// TIA Portal V20 export
ORGANIZATION_BLOCK "Startup"   // OB1020, LAD, Startup
TITLE = "Complete Restart"
// stored: AutoNumber false, IsIECCheckEnabled true, Namespace Unit1.Em3, SetENOAutomatically true
   VAR_INPUT
      LostRetentive : Bool;   // True if retentive data are lost
      LostRTC : Bool;   // True if date and time are lost
   END_VAR
BEGIN

REGION Network 1 (SCL): Build the Absolut Reference Designator
   // Set the Absoult Reference Designator in the Config DB
   IF LEN(IN := "Unit1.Em3.Config".em.referenceDesignator.parent) <> 0 THEN
       "Unit1.Em3.Config".em.referenceDesignator.combined := CONCAT_WSTRING(IN1 := "Unit1.Em3.Config".em.referenceDesignator.parent, IN2 := WSTRING#'.', IN3 := "Unit1.Em3.Config".em.referenceDesignator.relative);
   ELSE
       "Unit1.Em3.Config".em.referenceDesignator.combined := "Unit1.Em3.Config".em.referenceDesignator.relative;
   END_IF;
END_REGION

REGION Network 2 (SCL): Assign axes data
   // This is an example how to assign axes to DB_ANY in DB Config. If you have axes, assign them here. The Config.axis[] variables will be handed over to the control modules. That enables a flexible programming.
   // Assign axes
   "Unit1.MotionNodes".PLCToMotion.TechnologyObject.Axis.MasterVirtual := "Unit1.Em3.Config".axis[1] := "BA010AZCR_MasterVirtualAxis";
   "Unit1.MotionNodes".PLCToMotion.TechnologyObject.Axis.UnwinderVirtual := "Unit1.Em3.Config".axis[2] := "BA010AZCR_UnwinderVirtualAxis";

   // FB Enable
   "Unit1.Em3.HmiInterface".cmMasterVirtualAxis.commands.enable := TRUE;
END_REGION

REGION Network 3 (SCL): CM Config
   // Master Virtual Axis
   "Unit1.Em3.Config".cmMasterVirtualAxis.referenceDesignator := WSTRING#'MasterVirtualAxis';
   "Unit1.Em3.Config".cmMasterVirtualAxis.disableAlarms := FALSE;
   "Unit1.Em3.Config".cmMasterVirtualAxis.masterControlPopUp := TRUE;

   // Unwinder Virtual Axis
   "Unit1.Em3.Config".cmUnwinderVirtualAxis.referenceDesignator := WSTRING#'UnwinderVirtualAxis';
   "Unit1.Em3.Config".cmUnwinderVirtualAxis.disableAlarms := FALSE;
   "Unit1.Em3.Config".cmUnwinderVirtualAxis.masterControlPopUp := TRUE;


   // Dancer Regulator
   "Unit1.Em3.Config".cmDancerRegulatorOnOff.referenceDesignator := WSTRING#'Dancer Regulator';
   "Unit1.Em3.Config".cmDancerRegulatorOnOff.monitoringLeavingFeedback := T#0MS;
   "Unit1.Em3.Config".cmDancerRegulatorOnOff.monitoringReachingFeedback := T#0MS;
   "Unit1.Em3.Config".cmDancerRegulatorOnOff.monitoringDiscrepancy := T#0ms;
   "Unit1.Em3.Config".cmDancerRegulatorOnOff.setOutputHomeContinuously := TRUE;
   "Unit1.Em3.Config".cmDancerRegulatorOnOff.setOutputWorkContinuously := TRUE;
   "Unit1.Em3.Config".cmDancerRegulatorOnOff.disableHomeCommand := FALSE;
   "Unit1.Em3.Config".cmDancerRegulatorOnOff.disableFeedbackHomePos := TRUE;
   "Unit1.Em3.Config".cmDancerRegulatorOnOff.disableFeedbackWorkPos := TRUE;
   "Unit1.Em3.Config".cmDancerRegulatorOnOff.disableAlarms := FALSE;
   "Unit1.Em3.Config".cmDancerRegulatorOnOff.resetOutputsOnError := FALSE;
   "Unit1.Em3.Config".cmDancerRegulatorOnOff.allwaysWaitOnReachingTime := FALSE;


   // Dancer Encoder
   "Unit1.Em3.Config".cmDancerEncoderAnalogInput.referenceDesignator := WSTRING#'Dancer Encoder';
   "Unit1.Em3.Config".cmDancerEncoderAnalogInput.physicalUnit := 'deg';
   "Unit1.Em3.Config".cmDancerEncoderAnalogInput.isUnipolarSignal := TRUE;
   "Unit1.Em3.Config".cmDancerEncoderAnalogInput.default := 0;
   "Unit1.Em3.Config".cmDancerEncoderAnalogInput.limitHigh2 := 20;
   "Unit1.Em3.Config".cmDancerEncoderAnalogInput.limitHigh1 := 15;
   "Unit1.Em3.Config".cmDancerEncoderAnalogInput.limitLow1 := -15;
   "Unit1.Em3.Config".cmDancerEncoderAnalogInput.limitLow2 := -20;
   "Unit1.Em3.Config".cmDancerEncoderAnalogInput.processValueMax := 43;
   "Unit1.Em3.Config".cmDancerEncoderAnalogInput.processValueMin := -43;
   "Unit1.Em3.Config".cmDancerEncoderAnalogInput.scaleAnalogUppPoint := 27648;
   "Unit1.Em3.Config".cmDancerEncoderAnalogInput.scaleAnalogLowPoint := 0;
   "Unit1.Em3.Config".cmDancerEncoderAnalogInput.scaleProcessUppPoint := 43;
   "Unit1.Em3.Config".cmDancerEncoderAnalogInput.scaleProcessLowPoint := -43;
   "Unit1.Em3.Config".cmDancerEncoderAnalogInput.disableAlarms := FALSE;


   // Dancer Electro Pneumatic Regulator
   "Unit1.Em3.Config".cmDancerElectroPneumaticRegulatorAnalogOutput.referenceDesignator := WSTRING#'Dancer Regulator';
   "Unit1.Em3.Config".cmDancerElectroPneumaticRegulatorAnalogOutput.physicalUnit := 'MPa';
   "Unit1.Em3.Config".cmDancerElectroPneumaticRegulatorAnalogOutput.isUnipolarSignal := TRUE;
   "Unit1.Em3.Config".cmDancerElectroPneumaticRegulatorAnalogOutput.default := 0;
   "Unit1.Em3.Config".cmDancerElectroPneumaticRegulatorAnalogOutput.limitHigh2 := 90;
   "Unit1.Em3.Config".cmDancerElectroPneumaticRegulatorAnalogOutput.limitHigh1 := 80;
   "Unit1.Em3.Config".cmDancerElectroPneumaticRegulatorAnalogOutput.limitLow1 := -80;
   "Unit1.Em3.Config".cmDancerElectroPneumaticRegulatorAnalogOutput.limitLow2 := -90;
   "Unit1.Em3.Config".cmDancerElectroPneumaticRegulatorAnalogOutput.processValueMax := 0.5;
   "Unit1.Em3.Config".cmDancerElectroPneumaticRegulatorAnalogOutput.processValueMin := 0.005;
   "Unit1.Em3.Config".cmDancerElectroPneumaticRegulatorAnalogOutput.scaleProcessUppPoint := 0.5;
   "Unit1.Em3.Config".cmDancerElectroPneumaticRegulatorAnalogOutput.scaleProcessLowPoint := 0.005;
   "Unit1.Em3.Config".cmDancerElectroPneumaticRegulatorAnalogOutput.scaleAnalogUppPoint := 27648;
   "Unit1.Em3.Config".cmDancerElectroPneumaticRegulatorAnalogOutput.scaleAnalogLowPoint := 0;
   "Unit1.Em3.Config".cmDancerElectroPneumaticRegulatorAnalogOutput.disableAlarms := TRUE;


   // Load Cell
   "Unit1.Em3.Config".cmLoadCellAnalogInput.referenceDesignator := WSTRING#'Load Cell AnalogInput';
   "Unit1.Em3.Config".cmLoadCellAnalogInput.physicalUnit := 'unit';
   "Unit1.Em3.Config".cmLoadCellAnalogInput.isUnipolarSignal := TRUE;
   "Unit1.Em3.Config".cmLoadCellAnalogInput.default := 0;
   "Unit1.Em3.Config".cmLoadCellAnalogInput.limitHigh2 := 50;
   "Unit1.Em3.Config".cmLoadCellAnalogInput.limitHigh1 := 40;
   "Unit1.Em3.Config".cmLoadCellAnalogInput.limitLow1 := -80;
   "Unit1.Em3.Config".cmLoadCellAnalogInput.limitLow2 := -90;
   "Unit1.Em3.Config".cmLoadCellAnalogInput.processValueMax := 40;
   "Unit1.Em3.Config".cmLoadCellAnalogInput.processValueMin := 0;
   "Unit1.Em3.Config".cmLoadCellAnalogInput.scaleAnalogUppPoint := 27648;
   "Unit1.Em3.Config".cmLoadCellAnalogInput.scaleAnalogLowPoint := 0;
   "Unit1.Em3.Config".cmLoadCellAnalogInput.scaleProcessUppPoint := 50;
   "Unit1.Em3.Config".cmLoadCellAnalogInput.scaleProcessLowPoint := 0;
   "Unit1.Em3.Config".cmLoadCellAnalogInput.disableAlarms := FALSE;


   // Web Guide EPC
   "Unit1.Em3.Config".cmWebGuideEpc.referenceDesignator := WSTRING#'Web Guide Epc';
   "Unit1.Em3.Config".cmWebGuideEpc.hwID.EkrOut_Auto_Sp_Acp_HW_ID := "BA010AZCREPCC3~EkrOut_Auto_Sp_Acp_1";
   "Unit1.Em3.Config".cmWebGuideEpc.hwID.EkrOut_CAM_Data_HW_ID := "BA010AZCREPCC3~EkrOut_CAM_Data_1";
   "Unit1.Em3.Config".cmWebGuideEpc.hwID.EkrOut_CLS_Data_HW_ID := "BA010AZCREPCC3~EkrOut_CLS_Data_1";
   "Unit1.Em3.Config".cmWebGuideEpc.hwID.EkrOut_Guiding_edges_HW_ID := "BA010AZCREPCC3~EkrOut_Guiding_edges_1";
   "Unit1.Em3.Config".cmWebGuideEpc.hwID.EkrOut_HEADER_Data_HW_ID := "BA010AZCREPCC3~EkrOut_HEADER_Data_1";
   "Unit1.Em3.Config".cmWebGuideEpc.hwID.EkrOut_POS_unit_HW_ID := "BA010AZCREPCC3~EkrOut_POS_unit_1";
   "Unit1.Em3.Config".cmWebGuideEpc.hwID.EkrOut_SEN_Data_HW_ID := "BA010AZCREPCC3~EkrOut_SEN_Data_1";
   "Unit1.Em3.Config".cmWebGuideEpc.hwID.EkrOut_Servo_Center_HW_ID := "BA010AZCREPCC3~EkrOut_Servo_Center_1";
   "Unit1.Em3.Config".cmWebGuideEpc.hwID.EkrOut_Setpoint_HW_ID := "BA010AZCREPCC3~EkrOut_Setpoint_1";
   "Unit1.Em3.Config".cmWebGuideEpc.hwID.EkrOut_Web_width_HW_ID := "BA010AZCREPCC3~EkrOut_Web_width_1";
   "Unit1.Em3.Config".cmWebGuideEpc.hwID.EkrIn_Auto_Sp_Acp_HW_ID := "BA010AZCREPCC3~EkrIn_Auto_Sp_Acp_1";
   "Unit1.Em3.Config".cmWebGuideEpc.hwID.EkrIn_HEADER_Data_HW_ID := "BA010AZCREPCC3~EkrIn_HEADER_Data_1";
   "Unit1.Em3.Config".cmWebGuideEpc.hwID.EkrIn_POS_unit_HW_ID := "BA010AZCREPCC3~EkrIn_POS_unit_1";
   "Unit1.Em3.Config".cmWebGuideEpc.hwID.EkrIn_Setpoint_HW_ID := "BA010AZCREPCC3~EkrIn_Setpoint_1";
   "Unit1.Em3.Config".cmWebGuideEpc.hwID.EkrIn_Web_width_HW_ID := "BA010AZCREPCC3~EkrIn_Web_width_1";


   // Dancer Safety Pin Idle Position
   "Unit1.Em3.Config".cmDancerSafetyPinIdlePosition.referenceDesignator := WSTRING#'DigitalSignal';
   "Unit1.Em3.Config".cmDancerSafetyPinIdlePosition.onDelay := T#0ms;
   "Unit1.Em3.Config".cmDancerSafetyPinIdlePosition.offDelay := T#0ms;
   "Unit1.Em3.Config".cmDancerSafetyPinIdlePosition.default := FALSE;
   "Unit1.Em3.Config".cmDancerSafetyPinIdlePosition.invertProcessValue := FALSE;
   "Unit1.Em3.Config".cmDancerSafetyPinIdlePosition.disableAlarms := FALSE;
END_REGION
END_ORGANIZATION_BLOCK
